// TIA Portal V18 export
// export: Created 2026-06-08T16:32:20.3686707Z, ExportSetting WithDefaults, DisplayName Totally Integrated Automation Portal, DisplayVersion V18, DisplayName TIA Portal Openness, DisplayVersion V18, DisplayName TIA Portal Version Control Interface, DisplayVersion V18, DisplayName STEP 7 Professional, DisplayVersion V18, DisplayName STEP 7 Safety, DisplayVersion V18, DisplayName WinCC Professional, DisplayVersion V18
DATA_BLOCK "PICK_UP_LID_ROBOT_DB"   // DB11
VERSION : 0.1
// stored: AutoNumber true, InstanceOfName PICK_UP_LID_ROBOT, InstanceOfType FB
"PICK_UP_LID_ROBOT"
BEGIN
END_DATA_BLOCK
